// Mitsubishi GX Works2 project: 240507_timechart10_양음변환1   PLC: Q03UDV

PROGRAM MAIN
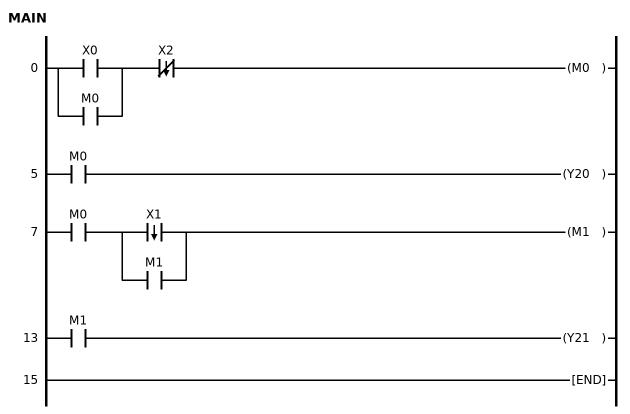
0     LD      X0
      OR      M0
      ANDFI   X2
      OUT     M0
5     LD      M0
      OUT     Y20
7     LD      M0
      LDF     X1
      OR      M1
      ANB
      OUT     M1
13    LD      M1
      OUT     Y21
15    END
END_PROGRAM
